TYPE ST_DummyRoomInputs :
STRUCT
    bButton : BOOL;
END_STRUCT
END_TYPE

(* stored: Version 1.1.0.1
   DUT ST_DummyRoomInputs: Id {0cfc25a1-9bd4-454d-abee-d575ec051344} *)
